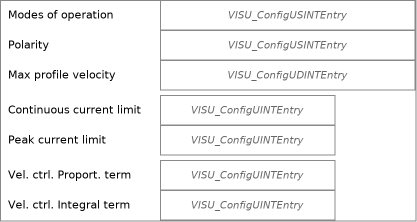
VISUALIZATION VISU_FaulhaberDriveConfig_Control  // 417x222
VAR_IN_OUT
	active : FaulhaberDriveConfig;
	editable : FaulhaberDriveConfig;
END_VAR
    Label (5,30 135x30), "Polarity"
    Frame (160,95 175x30)
        shows VISU_ConfigUINTEntry(active := active.continuousCurrentLimit, editable := editable.continuousCurrentLimit)
    Label (5,95 135x30), "Continuous current limit"
    Label (5,125 135x30), "Peak current limit"
    Frame (160,125 175x30)
        shows VISU_ConfigUINTEntry(active := active.peakCurrentLimit, editable := editable.peakCurrentLimit)
    Frame (160,160 175x30)
        shows VISU_ConfigUINTEntry(active := active.velocityControlProportionalTerm, editable := editable.velocityControlProportionalTerm)
    Label (5,160 135x30), "Vel. ctrl. Proport. term"
    Label (5,190 135x30), "Vel. ctrl. Integral term"
    Frame (160,190 175x30)
        shows VISU_ConfigUINTEntry(active := active.velocityControlIntegralTerm, editable := editable.velocityControlIntegralTerm)
    Label (5,0 135x30), "Modes of operation"
    Frame (160,0 255x30)
        shows VISU_ConfigUSINTEntry(active := active.modesOfOperation, editable := editable.modesOfOperation)
    Frame (160,30 255x30)
        shows VISU_ConfigUSINTEntry(active := active.polarity, editable := editable.polarity)
    Frame (160,60 255x30)
        shows VISU_ConfigUDINTEntry(active := active.maxProfileVelocity, editable := editable.maxProfileVelocity)
    Label (5,60 135x30), "Max profile velocity"
END_VISUALIZATION

(* stored: Version 1.1.0.1, ProductVersion 3.1.4019.2
   Visu VISU_FaulhaberDriveConfig_Control: Id {9b04152c-e67a-49b8-8d5b-29a4ab606fed} *)
